// TIA Portal project "Sandstrahlanlage" (V16)

(* hardware
DEVICE "S7300/ET200M-Station_1"  S7-300 station
   slot 0: "Profilschiene_0"  Rail  6ES7 390-1***0-0AA0
   slot 1: "PS 307 5A_1"  PS 307 5A  6ES7 307-1EA00-0AA0
   slot 2: "PLC_1"  CPU 314C-2 PN/DP  6ES7 314-6EH04-0AB0  V3.3
      slot 2: "PROFINET-Schnittstelle_1"  PN-IO
         slot 1: "Port_1"  Port
         slot 2: "Port_2"  Port
      slot 5: "DI 24/DO 16_1"  DI24/DO16
      slot 6: "AI 5/AO 2_1"  AI5/AO2
      slot 7: "Zählen_1"  Counter
      slot 8: "Positionieren_1"  Positioning
   slot 4: "DI 16/DO 16x24VDC/0.5A_1"  DI16/DO16 x 24V / 0.5A  6ES7 323-1BL00-0AA0
   slot 5: "CP 343-2P_1"  CP 343-2P  6GK7 343-2AH11-0XA0  V3.1
*)

// ===== PLC "PLC_1"  CPU 314C-2 PN/DP =====

FUNCTION_BLOCK "Automatic_Mode"   // FB1, FBD
{ S7_Optimized_Access := 'FALSE' }
VERSION : 0.1
   VAR_INPUT
      S2_Automatikbetrieb : Bool;
      S5_Halt : Bool;
      Endschalter_Tur_Unten : Bool;
      Grundstellung : Bool;
      Tur_Geschlossen : Bool;
      S4_Raupenband_Vor : Bool;
      S3_Ruckwarts : Bool;
      M_Steuerspannung : Bool;
      Takt : Bool;
   END_VAR
   VAR_OUTPUT
      M_Automatik_A : Bool;
      Lautewerk : Bool;
      Strahlmitteltransport : Bool;
      Strahlmittelzuteilung : Bool;
      Schwingforderrinne : Bool;
      Raupenband_Vor : Bool;
      Raupenband_Zuruck : Bool;
      Schleuderrad : Bool;
      Rundumleuchte : Bool;
      Tur_Schliessen : Bool;
   END_VAR
   VAR
      M_Automatik : Bool;
      Schritt_1 : Bool;
      Schritt_2 : Bool;
      Schritt_3 : Bool;
      Schritt_4 : Bool;
      Schritt_5 : Bool;
      Schritt_6 : Bool;
      M_Raupenband_vor : Bool;
      M_Rundumleuchte : Bool;
      M_Strahlmittelzuteilung : Bool;
      M_Schwingforderrinne : Bool;
      M_Strahlmitteltransport : Bool;
      M_Schleuderrad : Bool;
      Verzogerung : Bool;
      Verzogerung_1 : Bool;
      Verzogerung_2 : Bool;
      TON_0 : Bool;
      TON_1 : Bool;
      M_Erlaubnis_Raupenband_fahren : Bool;
      IEC_Timer_0_Instance : TON;
      IEC_Timer_0_Instance_1 : TON;
   END_VAR
BEGIN

REGION Network 1
   // Enabling the automatic mode
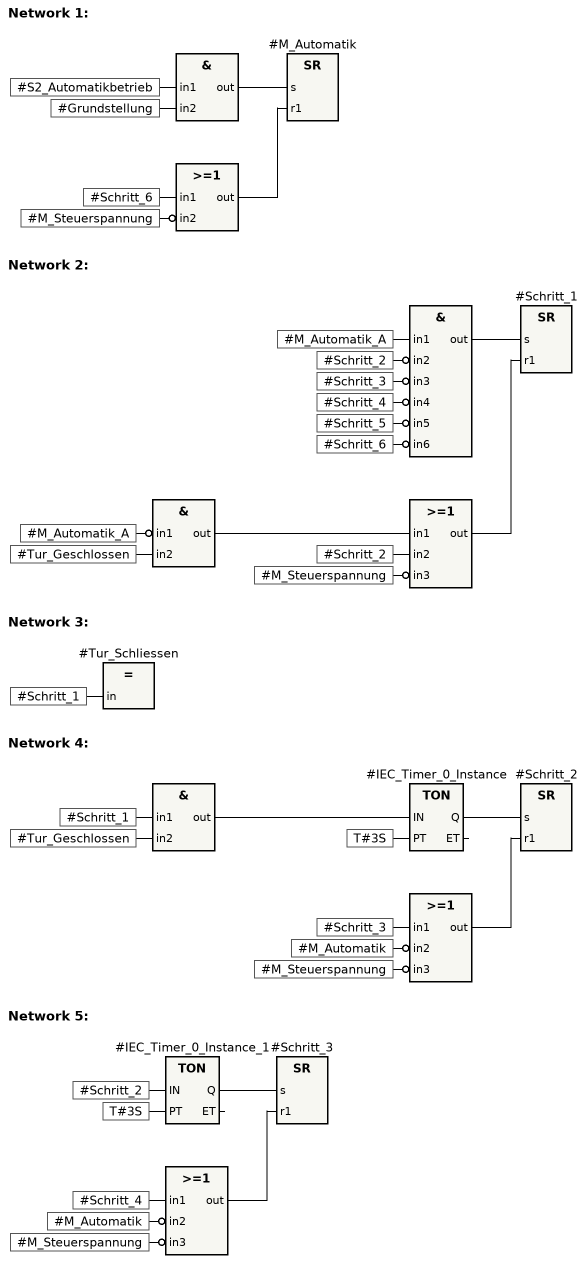
   IF #S2_Automatikbetrieb AND #Grundstellung THEN
       #M_Automatik := TRUE;   // SR flip-flop
   END_IF;
   IF #Schritt_6 OR NOT #M_Steuerspannung THEN #M_Automatik := FALSE; END_IF;
END_REGION

REGION Network 2
   // Sequencer. Step 1
   IF #M_Automatik_A AND NOT #Schritt_2 AND NOT #Schritt_3 AND NOT #Schritt_4 AND NOT #Schritt_5 AND NOT #Schritt_6 THEN
       #Schritt_1 := TRUE;   // SR flip-flop
   END_IF;
   IF (NOT #M_Automatik_A AND #Tur_Geschlossen) OR #Schritt_2 OR NOT #M_Steuerspannung THEN
       #Schritt_1 := FALSE;
   END_IF;
END_REGION

REGION Network 3
   #Tur_Schliessen := #Schritt_1;
END_REGION

REGION Network 4
   // Sequencer. Step 2
   #IEC_Timer_0_Instance.TON(IN := #Schritt_1 AND #Tur_Geschlossen, PT := T#3S);
   IF #IEC_Timer_0_Instance.Q THEN
       #Schritt_2 := TRUE;   // SR flip-flop
   END_IF;
   IF #Schritt_3 OR NOT #M_Automatik OR NOT #M_Steuerspannung THEN #Schritt_2 := FALSE; END_IF;
END_REGION

REGION Network 5
   // Sequencer. Step 3
   #IEC_Timer_0_Instance_1.TON(IN := #Schritt_2, PT := T#3S);
   IF #IEC_Timer_0_Instance_1.Q THEN
       #Schritt_3 := TRUE;   // SR flip-flop
   END_IF;
   IF #Schritt_4 OR NOT #M_Automatik OR NOT #M_Steuerspannung THEN #Schritt_3 := FALSE; END_IF;
END_REGION

REGION Network 6
   // Sequencer. Step 4
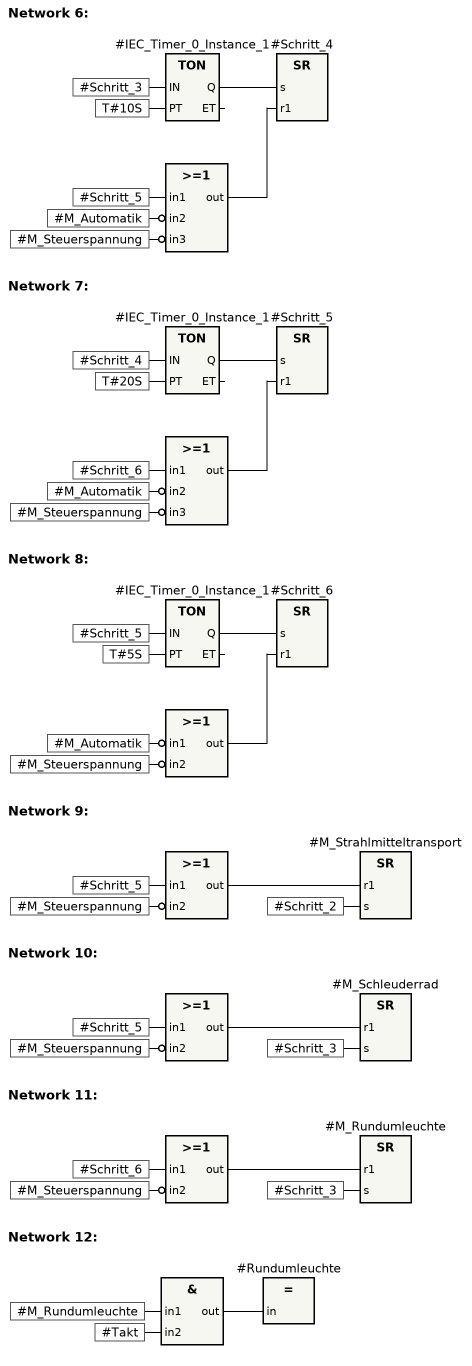
   #IEC_Timer_0_Instance_1.TON(IN := #Schritt_3, PT := T#10S);
   IF #IEC_Timer_0_Instance_1.Q THEN
       #Schritt_4 := TRUE;   // SR flip-flop
   END_IF;
   IF #Schritt_5 OR NOT #M_Automatik OR NOT #M_Steuerspannung THEN #Schritt_4 := FALSE; END_IF;
END_REGION

REGION Network 7
   // Sequencer. Step 5
   #IEC_Timer_0_Instance_1.TON(IN := #Schritt_4, PT := T#20S);
   IF #IEC_Timer_0_Instance_1.Q THEN
       #Schritt_5 := TRUE;   // SR flip-flop
   END_IF;
   IF #Schritt_6 OR NOT #M_Automatik OR NOT #M_Steuerspannung THEN #Schritt_5 := FALSE; END_IF;
END_REGION

REGION Network 8
   // Sequencer. Step 6
   #IEC_Timer_0_Instance_1.TON(IN := #Schritt_5, PT := T#5S);
   IF #IEC_Timer_0_Instance_1.Q THEN
       #Schritt_6 := TRUE;   // SR flip-flop
   END_IF;
   IF NOT #M_Automatik OR NOT #M_Steuerspannung THEN #Schritt_6 := FALSE; END_IF;
END_REGION

REGION Network 9
   IF #Schritt_2 THEN
       #M_Strahlmitteltransport := TRUE;   // SR flip-flop
   END_IF;
   IF #Schritt_5 OR NOT #M_Steuerspannung THEN #M_Strahlmitteltransport := FALSE; END_IF;
END_REGION

REGION Network 10
   IF #Schritt_3 THEN
       #M_Schleuderrad := TRUE;   // SR flip-flop
   END_IF;
   IF #Schritt_5 OR NOT #M_Steuerspannung THEN #M_Schleuderrad := FALSE; END_IF;
END_REGION

REGION Network 11
   IF #Schritt_3 THEN
       #M_Rundumleuchte := TRUE;   // SR flip-flop
   END_IF;
   IF #Schritt_6 OR NOT #M_Steuerspannung THEN #M_Rundumleuchte := FALSE; END_IF;
END_REGION

REGION Network 12
   #Rundumleuchte := #M_Rundumleuchte AND #Takt;
END_REGION

REGION Network 13
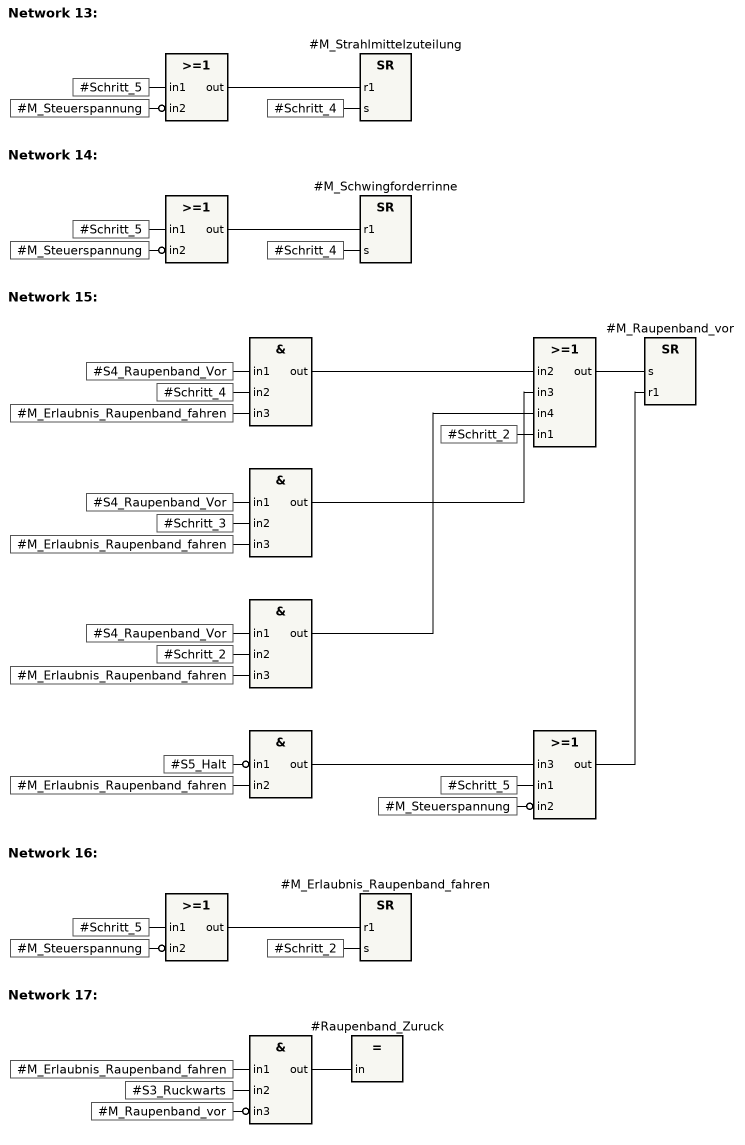
   IF #Schritt_4 THEN
       #M_Strahlmittelzuteilung := TRUE;   // SR flip-flop
   END_IF;
   IF #Schritt_5 OR NOT #M_Steuerspannung THEN #M_Strahlmittelzuteilung := FALSE; END_IF;
END_REGION

REGION Network 14
   IF #Schritt_4 THEN
       #M_Schwingforderrinne := TRUE;   // SR flip-flop
   END_IF;
   IF #Schritt_5 OR NOT #M_Steuerspannung THEN #M_Schwingforderrinne := FALSE; END_IF;
END_REGION

REGION Network 15
   IF (#S4_Raupenband_Vor AND #Schritt_4 AND #M_Erlaubnis_Raupenband_fahren) OR (#S4_Raupenband_Vor AND #Schritt_3 AND #M_Erlaubnis_Raupenband_fahren) OR (#S4_Raupenband_Vor AND #Schritt_2 AND #M_Erlaubnis_Raupenband_fahren) OR #Schritt_2 THEN
       #M_Raupenband_vor := TRUE;   // SR flip-flop
   END_IF;
   IF (NOT #S5_Halt AND #M_Erlaubnis_Raupenband_fahren) OR #Schritt_5 OR NOT #M_Steuerspannung THEN
       #M_Raupenband_vor := FALSE;
   END_IF;
END_REGION

REGION Network 16
   IF #Schritt_2 THEN
       #M_Erlaubnis_Raupenband_fahren := TRUE;   // SR flip-flop
   END_IF;
   IF #Schritt_5 OR NOT #M_Steuerspannung THEN #M_Erlaubnis_Raupenband_fahren := FALSE; END_IF;
END_REGION

REGION Network 17
   #Raupenband_Zuruck := #M_Erlaubnis_Raupenband_fahren AND #S3_Ruckwarts AND NOT #M_Raupenband_vor;
END_REGION
END_FUNCTION_BLOCK

ORGANIZATION_BLOCK "Main"   // OB1, LAD
TITLE = "Main Program Sweep (Cycle)"
{ S7_Optimized_Access := 'FALSE' }
VERSION : 0.1
   VAR_TEMP
      OB1_EV_CLASS : Byte;   // Bits 0-3 = 1 (Coming event), Bits 4-7 = 1 (Event class 1)
      OB1_SCAN_1 : Byte;   // 1 (Cold restart scan 1 of OB 1), 3 (Scan 2-n of OB 1)
      OB1_PRIORITY : Byte;   // Priority of OB Execution
      OB1_OB_NUMBR : Byte;   // 1 (Organization block 1, OB1)
      OB1_RESERVED_1 : Byte;   // Reserved for system
      OB1_RESERVED_2 : Byte;   // Reserved for system
      OB1_PREV_CYCLE : Int;   // Cycle time of previous OB1 scan (milliseconds)
      OB1_MIN_CYCLE : Int;   // Minimum cycle time of OB1 (milliseconds)
      OB1_MAX_CYCLE : Int;   // Maximum cycle time of OB1 (milliseconds)
      OB1_DATE_TIME : Date_And_Time;   // Date and time OB1 started
   END_VAR
BEGIN
END_ORGANIZATION_BLOCK